Staubli VAL3: remote_loadHome.pgx

program remote_loadHome(num& x_nResult[] (dimensions=1))
begin
  //
  // INIT
  //
  cycleStatus:bHomeLoaded=false
  // load the home home
  x_nResult=jHome:libLoad(saveData:sPathTraj+"HOME")
  if x_nResult==0
    // home loaded
    cycleStatus:bHomeLoaded=true
    //
  endIf
  //
end
